FUNCTION_BLOCK ServoNC EXTENDS FBA_TrifectaDrive IMPLEMENTS I_EncodedDrive
VAR_OUTPUT	
	ready : BOOL;
	position : LREAL;
	velocity : LREAL;
END_VAR
VAR
	axis : AXIS_REF;
	
	mcReadPosition : MC_ReadActualPosition; //continuous enable FBs
	mcReadVelocity : MC_ReadActualVelocity;
	mcReadError : MC_ReadAxisError;
	mcPower : MC_Power;
	
	mcReset : MC_Reset; //rising edge FBs
	mcMoveAbsolute : MC_MoveAbsolute;
	mcMoveRelative : MC_MoveRelative;
	mcMoveVelocity : MC_MoveVelocity;
	
	mcSetPosition : MC_SetPosition;
	mcStop : MC_Stop;
END_VAR
VAR_STAT CONSTANT
	targetingVelocity : INT := 500;
	continuousVelocity : INT := 100;
END_VAR

override();

blocks();

mcReset.Execute := FALSE;
mcMoveAbsolute.Execute := FALSE;
mcMoveRelative.Execute := FALSE;
mcMoveVelocity.Execute := FALSE;
mcSetPosition.Execute := FALSE;
mcStop.Execute := FALSE;

blocks();

ready := bEnable AND NOT Active AND HomeSet;

PROPERTY Active : BOOL
GET
Active := 
	mcMoveAbsolute.Busy OR 
	mcMoveRelative.Busy OR 
	mcMoveVelocity.Busy OR 
	mcSetPosition.Busy OR 
	mcReset.Busy OR 
	mcStop.Busy OR 
	step <> 0;
END_GET
END_PROPERTY

METHOD PRIVATE blocks : BOOL
mcReadPosition(
	Axis:= axis, 
	Enable:= TRUE, 
	Valid=> , 
	Busy=> , 
	Error=> , 
	ErrorID=> , 
	Position=> position);
	
mcReadVelocity(
	Axis:= axis, 
	Enable:= TRUE, 
	Valid=> , 
	Busy=> , 
	Error=> , 
	ErrorID=> , 
	ActualVelocity=> velocity);
	
mcReadError(
	Axis:= axis, 
	Enable:= TRUE, 
	Valid=> , 
	Busy=> , 
	Error=> , 
	ErrorID=> , 
	AxisErrorID=> );

mcReset(
	Axis:= axis, 
	Execute:= , 
	Done=> , 
	Busy=> , 
	Error=> , 
	ErrorID=> );

mcPower(
	Axis:= axis, 
	Enable:= bEnable, 
	Enable_Positive:= TRUE, 
	Enable_Negative:= TRUE, 
	Override:= 100, 
	BufferMode:= , 
	Options:= , 
	Status=> , 
	Busy=> , 
	Active=> , 
	Error=> , 
	ErrorID=> );

mcMoveAbsolute(
	Axis:= axis, 
	Execute:= , 
	Position:= , 
	Velocity:= targetingVelocity, 
	Acceleration:= , 
	Deceleration:= , 
	Jerk:= , 
	BufferMode:= , 
	Options:= , 
	Done=> , 
	Busy=> , 
	Active=> , 
	CommandAborted=> , 
	Error=> , 
	ErrorID=> );
	
mcMoveRelative(
	Axis:= axis, 
	Execute:= , 
	Distance:= ,
	Velocity:= targetingVelocity, 
	Acceleration:= , 
	Deceleration:= , 
	Jerk:= , 
	BufferMode:= , 
	Options:= , 
	Done=> , 
	Busy=> , 
	Active=> , 
	CommandAborted=> , 
	Error=> , 
	ErrorID=> );
	
mcMoveVelocity( //stopped with stop();
	Axis:= axis, 
	Execute:= , 
	Velocity:= continuousVelocity, 
	Acceleration:= , 
	Deceleration:= , 
	Jerk:= , 
	Direction:= , 
	BufferMode:= , 
	Options:= , 
	InVelocity=> , 
	Busy=> , 
	Active=> , 
	CommandAborted=> , 
	Error=> , 
	ErrorID=> );
	
mcSetPosition(
	Axis:= axis, 
	Execute:= , 
	Position:= , 
	Mode:= , 
	Options:= , 
	Done=> , 
	Busy=> , 
	Error=> , 
	ErrorID=> );
	
mcStop(
	Axis:= axis, 
	Execute:= , 
	Deceleration:= , 
	Jerk:= , 
	Options:= , 
	Done=> , 
	Busy=> , 
	Active=> , 
	CommandAborted=> , 
	Error=> , 
	ErrorID=> );
END_METHOD

PROPERTY CurrentPosition : LREAL
GET
CurrentPosition := position;
END_GET
SET
position := CurrentPosition;
END_SET
END_PROPERTY

PROPERTY Error : BOOL
GET
error := 
	mcMoveAbsolute.Error OR 
	mcMoveRelative.Error OR 
	mcMoveVelocity.Error OR 
	mcSetPosition.Error OR 
	mcReset.Error OR 
	mcStop.Error OR
	mcReadError.AxisErrorID > 0;
END_GET
END_PROPERTY

METHOD homingSequence : BOOL
CASE step OF
	Homing.IDLE:
		reset();
		IF bEnable THEN
			step := Homing.START;
		END_IF
		
	Homing.START:
		IF AtHome THEN
			mcMoveVelocity.Execute := FALSE;
			step := Homing.STOP;
			
		ELSIF AtInnerLimit THEN
			mcMoveVelocity.Execute := FALSE;
			step := Homing.RETRY;
			
		ELSE
			mcMoveVelocity.Direction := MC_Negative_Direction;
			mcMoveVelocity.Execute := NOT mcMoveVelocity.Execute;
		END_IF
		
	Homing.RETRY:
		IF AtOuterLimit THEN
			mcMoveVelocity.Execute := FALSE;
			step := Homing.START;
		ELSE
			mcMoveVelocity.Direction := MC_Positive_Direction;
			mcMoveVelocity.Execute := NOT mcMoveVelocity.Execute;
		END_IF
		
	Homing.STOP:
		IF velocity = 0 THEN
			mcStop.Execute := FALSE;
			step := Homing.SET;
		ELSE
			mcStop.Execute := TRUE;
		END_IF
		
	Homing.SET:
		IF position = 0 THEN
			mcSetPosition.Execute := FALSE;
			homingSequence := TRUE;
			step := Homing.DONE;
		ELSE
			mcSetPosition.Position := 0;
			mcSetPosition.Execute := TRUE;
		END_IF
		
	Homing.DONE:
		homingComplete := TRUE;
		step := Homing.IDLE;
		
END_CASE
END_METHOD

METHOD moveAbsolute : BOOL
VAR_INPUT
	newTarget : LREAL;
END_VAR
(*
VAR_OUTPUT
	fault : BOOL;
END_VAR
*)
IF NOT Active AND NOT error THEN
	mcMoveAbsolute.Position := newTarget;
	mcMoveAbsolute.Execute := TRUE;
END_IF

moveAbsolute := (*mcMoveAbsolute.Done AND mcMoveAbsolute.Active;*)
	position = newTarget;
END_METHOD

METHOD moveContinuous : BOOL
VAR_INPUT
	//direction : BOOL; //direction (F = inwards, T = outwards)
	direction : MC_Direction;
END_VAR
(*
IF mcMoveVelocity.Active THEN
	stop();
END_IF

IF NOT mcStop.Done THEN
	RETURN;
END_IF
*)
(*
IF direction THEN
	mcMoveVelocity.Direction := MC_Positive_Direction;
ELSE
	mcMoveVelocity.Direction := MC_Negative_Direction;
END_IF
*)
mcMoveVelocity.Direction := direction;

IF NOT mcMoveVelocity.Error THEN
	mcMoveVelocity.Execute := TRUE;
	moveContinuous := TRUE;
END_IF
END_METHOD

METHOD moveRelative : BOOL
VAR_INPUT
	distance : LREAL;
END_VAR
mcMoveRelative.Distance := distance;

moveRelative := mcMoveRelative.Done;
END_METHOD

METHOD PRIVATE override : BOOL
VAR_INPUT
END_VAR
(*
-at home and attempting to traverse outward
-at outer limit and attempting to traverse outward
-at inner limit and attempting to traverse inwards
*)
(*
inward = negative direction, negative velocity
outward = positive direction, positive velocity
*)

IF error THEN
	stop();
	reset();
	
ELSIF
	AtHome AND (TargetPosition > CurrentPosition OR velocity > 0) OR
	AtInnerLimit AND (TargetPosition > CurrentPosition OR velocity > 0) OR
	AtOuterLimit AND (TargetPosition < CurrentPosition OR velocity < 0)
THEN
	stop();
END_IF
END_METHOD

METHOD reset : BOOL
VAR_INPUT
END_VAR
mcReset.Execute := TRUE;

reset := mcReset.Done;
END_METHOD

METHOD stop : BOOL
VAR_INPUT
END_VAR
mcStop.Execute := TRUE;

mcMoveAbsolute.Execute := FALSE;
mcMoveRelative.Execute := FALSE;
mcMoveVelocity.Execute := FALSE;
END_METHOD

PROPERTY TargetPosition : LREAL
GET
END_GET
SET
moveAbsolute(newTarget := TargetPosition);
END_SET
END_PROPERTY

METHOD toHome : BOOL
VAR_INPUT
END_VAR
moveAbsolute(newTarget := 0);

toHome := AtHome;
END_METHOD

END_FUNCTION_BLOCK

(* stored: Version 1.1.0.1, ProductVersion 3.1.4024.11
   POU ServoNC: Id {4b82acd5-b43d-4437-930d-dd2d54682ea9}, SpecialFunc None
   Folder Private: Id {d6909568-bb93-45b7-82f2-cda1f893b190}
   Folder Properties: Id {fcd2e297-efca-46b4-96d8-07d1b7e7f038}
   Property Active: Id {fd93c0eb-b26b-44ed-a853-733964aa4dfc}
   Get Get: Id {732094d8-57e9-4263-82a2-a9ce9f969abb}
   Method blocks: Id {66e3a405-e872-4f52-b1b9-79f0c704f2a3}
   Property CurrentPosition: Id {67266511-06ee-405a-a5e7-79a2f88ccedf}
   Get Get: Id {e14867d2-b9e4-417e-871c-d699129b9dbf}
   Set Set: Id {166142fe-00c4-4e1d-bfa5-87cb8ff8700c}
   Property Error: Id {7e6ecac9-383f-431a-a546-cdf37505bd2c}
   Get Get: Id {22f0f866-23d1-446a-ad85-9990d8a446d7}
   Method homingSequence: Id {9801e5c2-0a6f-4ef0-ab5d-196ce8d10e7c}
   Method moveAbsolute: Id {1b14f767-77c4-41d0-8625-24688ac4d67d}
   Method moveContinuous: Id {b32535c3-6521-4e64-8d0e-cdab1af59453}
   Method moveRelative: Id {903dcbc7-8ba3-464b-81c8-4ae416934fdf}
   Method override: Id {a1a7b4c9-7e4c-4f10-97ee-2fce3b812262}
   Method reset: Id {b3c46065-9d19-4b54-adcf-2aa2d7909347}
   Method stop: Id {37bbe6c8-de36-4347-81d3-a6f7bd19dd38}
   Property TargetPosition: Id {ad8a2367-abf9-4f2d-b4a6-4788c3fdc41d}
   Get Get: Id {9005c10f-2d8b-485d-b1e1-3323ccbe71a3}
   Set Set: Id {c76d9784-3e46-4032-9f1d-eba0a54c9f4e}
   Method toHome: Id {23d0a0c3-9473-4538-9331-0e0f23d646a2} *)
